// TIA Portal V17 export
// export: Created 2022-07-28T18:03:20.5825143Z, ExportSetting None, DisplayName Totally Integrated Automation Portal, DisplayVersion V17, DisplayName TIA Portal Openness, DisplayVersion V17, DisplayName TIA Portal Teamcenter Gateway, DisplayVersion V17, DisplayName TIA Portal Version Control Interface, DisplayVersion V17, DisplayName TIA Portal Test Suite Advanced, DisplayVersion V17, DisplayName SINAMICS Startdrive Advanced, DisplayVersion V17, DisplayName SINAMICS DCC, DisplayVersion V17, DisplayName SINAMICS Startdrive G130, G150, S120, S150, SINAMICS MV, S210, DisplayVersion V17, DisplayName SINAMICS Startdrive G110M, G120, G120C, G120D, G120P, G115D, DisplayVersion V17, DisplayName STEP 7 Professional, DisplayVersion V17, DisplayName SIMATIC Energy Suite, DisplayVersion V17, DisplayName STEP 7 CFC, DisplayVersion V17, DisplayName STEP 7 Safety, DisplayVersion V17, DisplayName WinCC Advanced / Unified PC, DisplayVersion V17, DisplayName SIMATIC Visualization Architect, DisplayVersion V17
TYPE "Lib_UDT_PID_Cascad_HMI"
   STRUCT
      i_ID { S7_SetPoint := 'True'} : Int;
      i_CLSID { S7_SetPoint := 'True'} : Int;
      i_CMD : Int;
      Config { S7_SetPoint := 'True'} : "_PID_Cascad_Config";
      Counters { ExternalWritable := 'False'; S7_SetPoint := 'True'} : "_PID_Cascad_Counters";   // Лічильники
      Status { ExternalWritable := 'False'} : "_PID_Cascad_StateHMI";
   END_STRUCT;
END_TYPE
